TYPE E_Type_Tache :	// Appel des différentes tâches que le robot va faire
(
	eAttendre, eDeplacement, eAction, eFinParcours
);
END_TYPE

(* stored: Version 1.1.0.1, ProductVersion 3.1.4024.11
   DUT E_Type_Tache: Id {c955f85a-845c-473e-b66d-c83b67f58550} *)
